{attribute 'obsolete' := 'DUT_MotionStage has been renamed to ST_MotionStage'}
TYPE DUT_MotionStage : ST_MotionStage; END_TYPE

(* stored: Version 1.1.0.1
   DUT DUT_MotionStage: Id {d370719e-8c1e-449e-9592-4ea6f820eba7} *)
